Fanuc KAREL source: ka00142.KL

PROGRAM KA00142
%STACKSIZE=65535
%PRIORITY=65535
%NOLOCKGROUP
-- UNRESOLVED DECLARATIONS (source type spelling not recovered)
-- SRC : ARRAY[2] OF TYPE_0x0017 (type_u16=0x2017)
-- DST : TYPE_0x001C (type_u16=0x001C)
BEGIN
-- UNRESOLVED_PC line 7 opcodes [2E 22 9D 33 B4] marker_code=0
-- UNRESOLVED_PC line 8 opcodes [22 9D 33 B3 23] marker_code=19
END KA00142
